Fanuc KAREL source: kt00643.KL

-- PROVISIONAL review KL for V770-1; original PC SHA256 a12e4e8b00025d83c8462ae7d3b4281a33a16a93f98e62ca32761508cebeab41
-- Incomplete behavior may be omitted. Consult companion uncertainty JSON. Do not deploy.
PROGRAM KT00643
%NOLOCKGROUP
VAR
  OUT : INTEGER
-- UNRESOLVED_DECL H1 type=002017
-- UNRESOLVED_DECL H2 type=002017
BEGIN
  -- UNRESOLVED_PC offsets 5-19; opcodes 2E,22,9D,33,B4
  -- UNRESOLVED_PC offsets 24-38; opcodes 2E,22,9D,33,B4
  -- UNRESOLVED_PC offsets 43-57; opcodes 2E,22,9D,33,B4
  -- UNRESOLVED_PC offsets 62-76; opcodes 2E,22,9D,33,B4
  -- UNRESOLVED_PC offsets 81-97; opcodes 22,9D,33,B3,48,23
  -- UNRESOLVED_PC offsets 102-106; opcodes 7F
END KT00643
